// TwinCAT 3 PLC project auto_fault_reset
// ProgramVersion: 3.1.4022.4
// libraries:
//   Tc2_ControllerToolbox, * (Beckhoff Automation GmbH)
//   Tc2_EtherCAT, * (Beckhoff Automation GmbH)
//   Tc2_MC2, * (Beckhoff Automation GmbH)
//   Tc2_Standard, * (Beckhoff Automation GmbH)
//   Tc2_System, * (Beckhoff Automation GmbH)
//   Tc3_Module, * (Beckhoff Automation GmbH)
//   VisuSymbols,3.5.10.0,System
// project tree:
//   / GlobalTextList.TcGTLO, PlcTask.TcTTO, Visualization Manager.TcVMO (not stored)
//   GVLs/ GVL.TcGVL
//   POUs/ MAIN.TcPOU, FB_TIMER.TcPOU
//   VISUs/ OpMode.TcTLO, Visualization.TcVIS
// real-time tasks:
//   TASK PlcTask: cycle T#10ms, priority 20, ADS port 350
// motion (NC):
//   TASK NC-Task 1 SAF: cycle T#2ms, priority 4, ADS port 501
//   TASK NC-Task 1 SVB: cycle T#10ms, priority 8, ADS port 511
//   AXIS Axis 1 (id 2)
//     OtherSettings: AllowMotionCmdToSlave=true
//     encoder EncType=19
//       EncPara: MaxCount=#x0fffffff
//         Inc: RefSoftSyncMask=#x03ffffff
//     drive DrvType=16
//       DrvPara: MaxCount=#xffffffff
//         Analog: ScaleFactorActTorque=0.1
//         TimeComp: TaskDelayCycles=1
//     controller CtrType=1
//       CtrPara: PriorControlFactor=1
//         PosDiffControl: Enable=false, Range=1000
//         Observer: BandWidth=20
//   AXIS Axis 2 (id 1)
//     Dynamic: Acceleration=500
//     Velo: SlowManual=10, FastManual=30
//     PositionAreaControl: Enable=false
//     TargetPosControl: Enable=false
//     OtherSettings: AllowMotionCmdToSlave=true
//     encoder EncType=19
//       EncPara: MaxCount=#xffffffff
//     drive DrvType=16
//       DrvPara: MaxCount=#xffffffff, DriveControlDWord=#x00020000
//         Analog: VeloReferenz=100, ScaleFactorActTorque=0.1
//         TimeComp: TaskDelayCycles=1
//     controller CtrType=1
//       CtrPara: PriorControlFactor=1
//         PosDiffControl: Enable=false
//         Observer: BandWidth=20
// I/O:
//   DEVICE Device 2 (EtherCAT), AmsNetId 192.168.101.251.3.1
//     Drive 1 (CiA402 Motor Control Device) [SOMANET CiA402 Drive]
// variable links:
//   NC-Task 1 SAF/Axes/Axis 2 <-> Device 2 (EtherCAT)/Drive 1 (CiA402 Motor Control Device)
//     Drive/Inputs/In/nDataIn3[0] <-> TxPDO Mapping 1/Torque actual value
//     Drive/Inputs/In/nState1 <-> TxPDO Mapping 1/Statusword
//     Drive/Inputs/In/nState2 <-> TxPDO Mapping 1/Statusword @bit 8
//     Drive/Inputs/In/nState4 @bit 1 <-> WcState/InputToggle
//     Drive/Inputs/In/nState4 <-> WcState/WcState
//     Drive/Inputs/In/nState5 <-> TxPDO Mapping 1/Modes of operation display
//     Drive/Outputs/Out/nCtrl1 <-> RxPDO Mapping 1/Controlword
//     Drive/Outputs/Out/nCtrl2 <-> RxPDO Mapping 1/Controlword @bit 8
//     Drive/Outputs/Out/nDataOut1 <-> RxPDO Mapping 1/Target position
//     Drive/Outputs/Out/nDataOut2 <-> RxPDO Mapping 1/Target velocity
//     Enc/Inputs/In/nDataIn1 <-> TxPDO Mapping 1/Position actual value
//     Enc/Inputs/In/nState4 @bit 1 <-> WcState/InputToggle
//     Enc/Inputs/In/nState4 <-> WcState/WcState
//   auto_fault_reset/auto_fault_reset Instance <-> Device 2 (EtherCAT)/Drive 1 (CiA402 Motor Control Device)
//     PlcTask Inputs/GVL.velocity_in <-> TxPDO Mapping 1/Velocity actual value
//     PlcTask Outputs/GVL.opmode <-> RxPDO Mapping 1/Modes of operation
//     PlcTask Outputs/GVL.torque_out <-> RxPDO Mapping 1/Target torque

CONFIGURATION auto_fault_reset
    RESOURCE PLC ON TwinCAT3
        TASK PlcTask(INTERVAL := T#10ms, PRIORITY := 20);
        PROGRAM MAIN WITH PlcTask : MAIN;
    END_RESOURCE
END_CONFIGURATION

// ---- GVLs/GVL.TcGVL
{attribute 'qualified_only'}
VAR_GLOBAL
	
	//OPMODE_CSP : SINT := 8;
	OPMODE_CSV : SINT := 9;
	OPMODE_CST : SINT := 10;
	
	OPMODE_STRINGS : ARRAY [1..2] OF STRING := ['CSV', 'CST']; 
	
	TARGET_AMPLITUDE : DINT := 100;
	SINUS_FREQUENCY : TIME := T#300MS; // Milliseconds
	AMPLITUDE_OFFSET : REAL := 0.0;

	
	RESET_HOLD_TIME : TIME := T#2S; // Reset time
	RESET_SIGNAL : TIME := T#10S; // Cycle time (Checks after n seconds for errors)

	velocity_in AT %I*:DINT;
	velocity_out AT %Q*: DINT;
	torque_out AT %Q*: INT;
	opmode AT %Q*: SINT := OPMODE_CST;
	
	NET_ID_CABINET : T_AmsNetID := '192.168.101.251.3.1';
	SLAVE_ADDR : UINT := 1001;
	OBJ_DIR_ERROR			: WORD := 16#203F;
	NO_ERROR : LINT := 16#20746C7561466F4E;
	STR_NO_ERROR : STRING := LINT_TO_STRING(NO_ERROR);
END_VAR

// ---- POUs/MAIN.TcPOU
PROGRAM MAIN
VAR
	timer : FB_TIMER();
	trigger : BOOL;
	busy: BOOL;
	errorID_sdo: UDINT;
	sdo_ret_value : LINT;
	
	check_for_error : BOOL := FALSE;
	reset_drive: BOOL;
	fbSdoRead       : FB_EcCoESdoRead;
	error : BOOL;
	
	state : UINT := 0;
	
	bStatusEnable : BOOL;
		// =============== Axis reference =========================
	AxisRef			: AXIS_REF;				// Axis reference (process data plc/nc)
	
	// =============== Motion function blocks =================
	fbMcPower 		: MC_Power;				// FB for enable and override
	fbMcReset 		: MC_Reset;				// FB to reset axis
	
	// Signal generator
	fbSignalGenerator : FB_CTRL_SIGNAL_GENERATOR;
	fManValue : REAL := 0;
	eMode : E_CTRL_MODE := eCTRL_MODE_ACTIVE;
	stParams : ST_CTRL_SIGNAL_GENERATOR_PARAMS;
	fOut : LREAL;
END_VAR

(*
Change in GVL (GVLs->GVL): 
	TARGET_AMPLITUDE_VELOCITY : DINT := 1000;
	SINUS_FREQUENCY : TIME := T#300MS; // Milliseconds
	AMPLITUDE_OFFSET : REAL := 0.0;

	RESET_HOLD_TIME : TIME := T#2S;
	RESET_SIGNAL : TIME := T#10S;
*)



CASE state OF
	0:
		// Init state
		fbMCPower(	Enable 			:= TRUE, 
			Enable_Positive	:= TRUE, 
			Enable_Negative	:= TRUE, 
			Override		:= 100.0,
			Axis			:= AxisRef,
			Status			=> bStatusEnable);
			
		fbMcReset(Execute := TRUE, Axis := AxisRef);
		stParams.eSignalType := eCTRL_SINUS;
		stParams.fAmplitude := GVL.TARGET_AMPLITUDE;
		stParams.fOffset := GVL.AMPLITUDE_OFFSET;
		stParams.tStart := T#0S;
		stParams.tCtrlCycleTime := T#1MS;
		stParams.tTaskCycleTime := T#1MS;
		stParams.tCylceDuration := GVL.SINUS_FREQUENCY; 
		state := 1;
	1:
		fbMcReset(Execute := FALSE, Axis := AxisRef);
		state := 2;
	
	2:
		// Execute state
		// Signal generator for velocity. 
		//stParams.fAmplitude := GVL.TARGET_AMPLITUDE;
		//fbSignalGenerator(fManValue := fManValue, eMode := eMode, fOut => fOut, stParams := stParams);
		//GVL.velocity_out := LREAL_TO_DINT(fOut);
		//GVL.torque_out := LREAL_TO_INT(fOut);
		//GVL.torque_out := 200;
		GVL.torque_out := DINT_TO_INT(GVL.TARGET_AMPLITUDE);
		IF eMode = eCTRL_MODE_RESET THEN
			eMode := eCTRL_MODE_ACTIVE;
		END_IF
	
		// Timer for error checking
		timer(trigger => trigger);
		
		IF trigger THEN
			check_for_error := TRUE;
		END_IF
		
		IF check_for_error THEN
			
			IF GVL.velocity_in < 40 THEN
				reset_drive := TRUE;
			END_IF
			
			// Read SDO Error Object
			fbSDORead(sNetId := GVL.NET_ID_CABINET,
					nSlaveAddr := GVL.SLAVE_ADDR, 
					nIndex := GVL.OBJ_DIR_ERROR, 
					nSubIndex := 1, 
					pDstBuf := ADR(sdo_ret_value), 
					cbBuflen := SIZEOF(sdo_ret_value), 
					bExecute := TRUE, 
					bError => error, 
					nErrId => errorID_sdo, 
					bBusy => busy);
			// If error value unequal zero, reset drive.		
			IF sdo_ret_value <> GVL.NO_ERROR THEN
				reset_drive := TRUE;
				// Reset signal generator
				eMode := eCTRL_MODE_RESET;					
			END_IF
				// Finish SDO Reading
				fbSDORead(sNetId := GVL.NET_ID_CABINET,
					nSlaveAddr := GVL.SLAVE_ADDR, 
					nIndex := GVL.OBJ_DIR_ERROR, 
					nSubIndex := 0, 
					pDstBuf := ADR(sdo_ret_value), 
					cbBuflen := SIZEOF(sdo_ret_value), 
					bExecute := FALSE, 
					bError => error, 
					nErrId => errorID_sdo, 
					bBusy => busy);
			check_for_error := FALSE;
		END_IF
		
		// Call reset functions
		// Reset Drive
		//F_DRIVE_RESET(reset_drive);
		// Reset NC Task
		fbMcReset(Execute := reset_drive, Axis := AxisRef);
		reset_drive := FALSE;
END_CASE

END_PROGRAM

// ---- POUs/FB_TIMER.TcPOU
FUNCTION_BLOCK FB_TIMER
VAR_INPUT
END_VAR
VAR_OUTPUT
	trigger: BOOL := FALSE;
END_VAR

VAR
	state_timer			: UINT := 0;
	t1 : TON();
	t2 : TON();
END_VAR

CASE state_timer OF
	0:
		t1.PT := GVL.RESET_HOLD_TIME; // Low
		t2.PT := GVL.RESET_SIGNAL; // High - Reset signal
		//t1.IN := TRUE;
		state_timer := 1;
	1:
		t2.PT := GVL.RESET_SIGNAL; // High - Reset signal
		t1();
		t2();
		t2.IN := NOT t1.Q;
		t1.IN := t2.Q;
		trigger := t2.Q;
END_CASE

END_FUNCTION_BLOCK

// ---- GlobalTextList.TcGTLO
TEXTLIST GlobalTextList
  62 = 'Op Mode'
  232 = 'Reset Cycle Time (in milliseconds)'
  915 = 'Reset Cycle Time (in seconds)'
  80 = 'Target Value (Position/Velocity/Torque'
END_TEXTLIST

// ---- VISUs/OpMode.TcTLO
TEXTLIST OpMode
  8 = 'CSP'
  9 = 'CSV'
  10 = 'CST'
   = ''
END_TEXTLIST

// ---- VISUs/Visualization.TcVIS
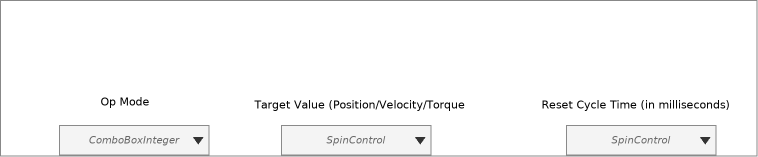
VISUALIZATION Visualization  // 758x157
    ComboBoxInteger (59,125 150x30), variable: GVL.opmode, text list: 'OpMode'
    SpinControl (281,125 150x30), variable: GVL.TARGET_AMPLITUDE
    Label (50,87 150x30), "Op Mode"
    Label (241,89 238x32), "Target Value (Position/Velocity/Torque"
    SpinControl (566,125 150x30), variable: GVL.RESET_SIGNAL
    Label (516,90 240x30), "Reset Cycle Time (in milliseconds)"
END_VISUALIZATION
